% RSLogix 500 project tank_alrams.RSS, saved by version 8.30.00.16 %
PROJECT "UNTITLED"    % processor: Bul.1763 MicroLogix 1100 Series B %

PROGRAM FILES
  LAD 2 "MAIN"  4 rungs
  LAD 3 "ALARMS"  7 rungs
  LAD 4 "IO"  4 rungs
  LAD 5 "CONTROLS"  6 rungs

DATA FILES
  O0 OUTPUT  7 elements
  I1 INPUT  13 elements
  S2 STATUS  66 elements
  B3 BINARY  1 elements
  T4 TIMER  4 elements
  C5 COUNTER  1 elements
  R6 CONTROL  1 elements
  N7 INTEGER  1 elements
  F8 FLOAT  1 elements

LADDER 2 "MAIN"
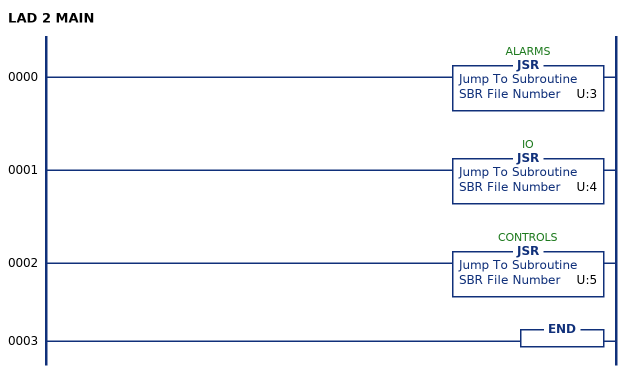
% Rung: 0 %
SOR JSR U:3 EOR
%   U:3  "ALARMS" %
% Rung: 1 %
SOR JSR U:4 EOR
%   U:4  "IO" %
% Rung: 2 %
SOR JSR U:5 EOR
%   U:5  "CONTROLS" %
% Rung: 3 %
SOR END EOR

LADDER 3 "ALARMS"
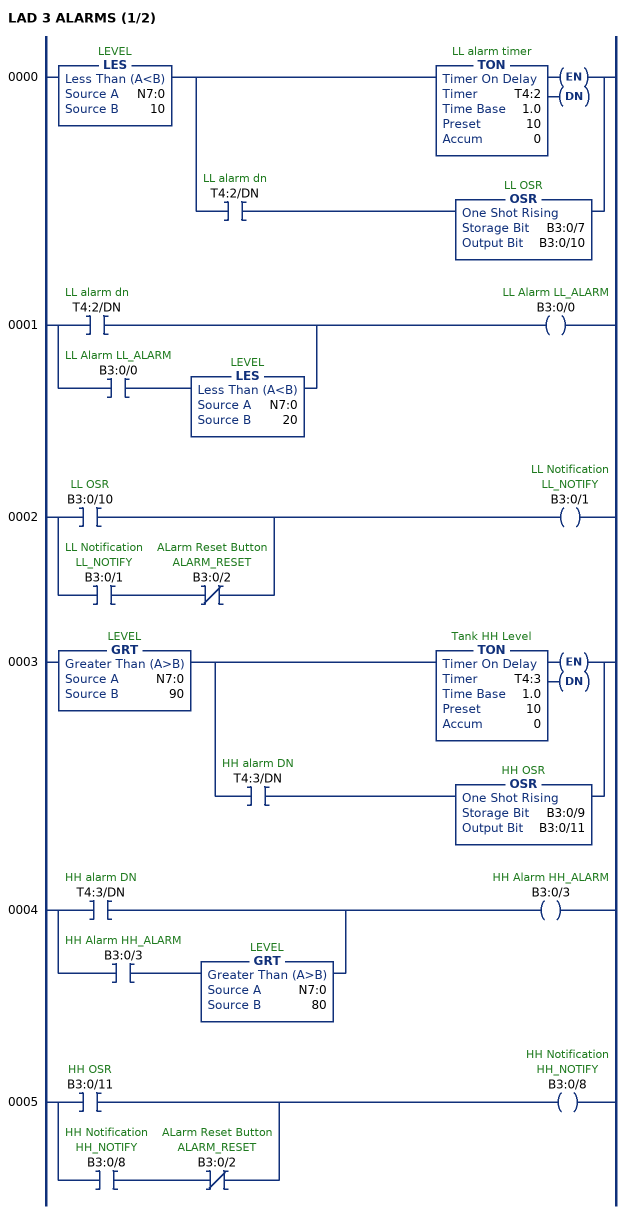
% Rung: 0 %
SOR LES N7:0 10 BST TON T4:2 1.0 10 0 NXB XIC T4:2/DN OSR B3:0/7 B3:0/10 BND EOR
%   N7:0  "LEVEL" %
%   T4:2  "LL alarm timer" %
%   T4:2/DN  "LL alarm dn" %
%   B3:0/7  "LL OSR" %
%   B3:0/10  "LL OSR" %
% Rung: 1 %
SOR BST XIC T4:2/DN NXB XIC B3:0/0 LES N7:0 20 BND OTE B3:0/0 EOR
%   T4:2/DN  "LL alarm dn" %
%   B3:0/0  LL_ALARM  "LL Alarm" %
%   N7:0  "LEVEL" %
% Rung: 2 %
SOR BST XIC B3:0/10 NXB XIC B3:0/1 XIO B3:0/2 BND OTE B3:0/1 EOR
%   B3:0/10  "LL OSR" %
%   B3:0/1  LL_NOTIFY  "LL Notification" %
%   B3:0/2  ALARM_RESET  "ALarm Reset Button" %
% Rung: 3 %
SOR GRT N7:0 90 BST TON T4:3 1.0 10 0 NXB XIC T4:3/DN OSR B3:0/9 B3:0/11 BND EOR
%   N7:0  "LEVEL" %
%   T4:3  "Tank HH Level" %
%   T4:3/DN  "HH alarm DN" %
%   B3:0/9  "HH OSR" %
%   B3:0/11  "HH OSR" %
% Rung: 4 %
SOR BST XIC T4:3/DN NXB XIC B3:0/3 GRT N7:0 80 BND OTE B3:0/3 EOR
%   T4:3/DN  "HH alarm DN" %
%   B3:0/3  HH_ALARM  "HH Alarm" %
%   N7:0  "LEVEL" %
% Rung: 5 %
SOR BST XIC B3:0/11 NXB XIC B3:0/8 XIO B3:0/2 BND OTE B3:0/8 EOR
%   B3:0/11  "HH OSR" %
%   B3:0/8  HH_NOTIFY  "HH Notification" %
%   B3:0/2  ALARM_RESET  "ALarm Reset Button" %

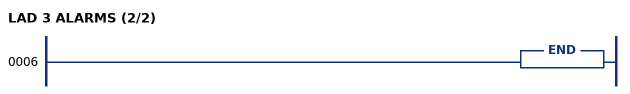
% Rung: 6 %
SOR END EOR

LADDER 4 "IO"
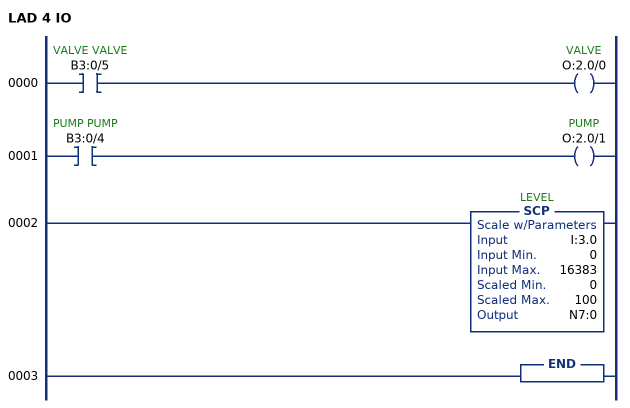
% Rung: 0 %
SOR XIC B3:0/5 OTE O:2.0/0 EOR
%   B3:0/5  VALVE  "VALVE" %
%   O:2.0/0  "VALVE" %
% Rung: 1 %
SOR XIC B3:0/4 OTE O:2.0/1 EOR
%   B3:0/4  PUMP  "PUMP" %
%   O:2.0/1  "PUMP" %
% Rung: 2 %
SOR SCP I:3.0 0 16383 0 100 N7:0 EOR
%   I:3.0  LEVEL  "LEVEL" %
%   N7:0  "LEVEL" %
% Rung: 3 %
SOR END EOR

LADDER 5 "CONTROLS"
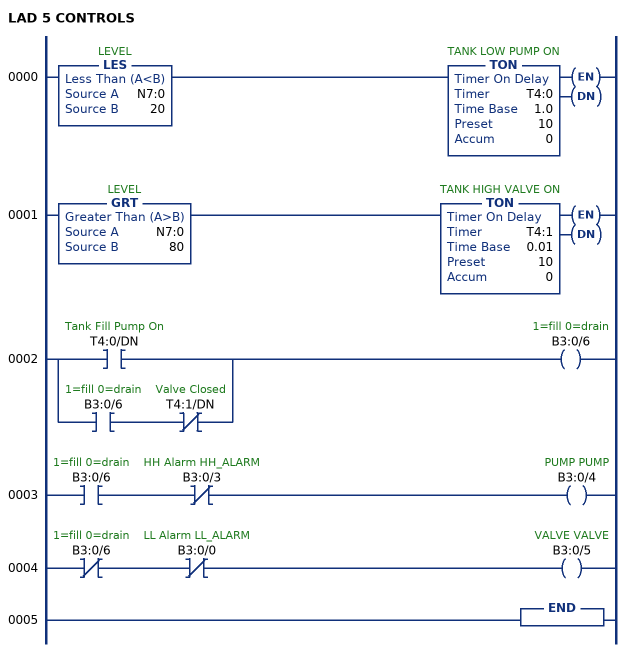
% Rung: 0 %
SOR LES N7:0 20 TON T4:0 1.0 10 0 EOR
%   N7:0  "LEVEL" %
%   T4:0  "TANK LOW PUMP ON" %
% Rung: 1 %
SOR GRT N7:0 80 TON T4:1 0.01 10 0 EOR
%   N7:0  "LEVEL" %
%   T4:1  "TANK HIGH VALVE ON" %
% Rung: 2 %
SOR BST XIC T4:0/DN NXB XIC B3:0/6 XIO T4:1/DN BND OTE B3:0/6 EOR
%   T4:0/DN  "Tank Fill Pump On" %
%   B3:0/6  "1=fill 0=drain" %
%   T4:1/DN  "Valve Closed" %
% Rung: 3 %
SOR XIC B3:0/6 XIO B3:0/3 OTE B3:0/4 EOR
%   B3:0/6  "1=fill 0=drain" %
%   B3:0/3  HH_ALARM  "HH Alarm" %
%   B3:0/4  PUMP  "PUMP" %
% Rung: 4 %
SOR XIO B3:0/6 XIO B3:0/0 OTE B3:0/5 EOR
%   B3:0/6  "1=fill 0=drain" %
%   B3:0/0  LL_ALARM  "LL Alarm" %
%   B3:0/5  VALVE  "VALVE" %
% Rung: 5 %
SOR END EOR

OTHER DOCUMENTED ADDRESSES
  O:2.0  "VALVE"
  O:2.1  "PUMP"

DATA TABLE (non-zero values as saved)
DATA T4
% .PRE .ACC %
% T4:0 % 10 0
% T4:1 % 10 0
% T4:2 % 10 0
% T4:3 % 10 0
